PROGRAM DataAcquisitionController
VAR
	// Handlers to call
	HandleOpcTagWriting : OpcTagWritingHandler;
	HandleMatlab 		: MatlabHandler;
	
	// Local variables
	_matlabBtn : BOOL;
	_matlabHmiValues : ST_MatlabValues;
END_VAR


HandleOpcTagWriting();

HandleMatlab(
			startButton := _matlabBtn,
			hmiValues => _matlabHmiValues);

PROPERTY MatlabBtn : BOOL
SET

_MatlabBtn := MatlabBtn;
END_SET
END_PROPERTY

PROPERTY MatlabHmiValues : ST_MatlabValues
GET

MatlabHmiValues := _matlabHmiValues;
END_GET
END_PROPERTY

END_PROGRAM

(* stored: Version 1.1.0.1, ProductVersion 3.1.4024.9
   POU DataAcquisitionController: Id {8ef7b23d-377f-464a-94da-dbf13a683f44}, SpecialFunc None
   Property MatlabBtn: Id {12390ade-eb97-4d4a-aa0b-dfac54f1b9cf}
   Set Set: Id {4570ab4c-2c20-47c1-93a4-d240137c3a55}
   Property MatlabHmiValues: Id {b30c06e2-1dce-4ae9-b5ea-96ee729b6002}
   Get Get: Id {0be0c361-5cc2-4877-86cc-6a7832ec5f7b} *)
